PROGRAM MAIN
VAR
	manual: Manual;
	automatic: Automatic;
	errorsAndWarnings: ErrorsWarnings;
END_VAR

IF gvl.ButtonGreen THEN
	gvl.MotorCompressor := TRUE;
ELSIF gvl.ButtonRed THEN
	gvl.MotorCompressor := FALSE;
END_IF

IF gvl.Switch THEN
	manual();
else
	automatic();
END_IF

errorsAndWarnings();

END_PROGRAM

(* stored: Version 1.1.0.1, ProductVersion 3.1.4024.12
   POU MAIN: Id {f07c1a1b-64dd-448f-b981-7b9317a5ba38}, SpecialFunc None *)
